SUBAPPLICATION Uebung_070 (* WBSD auf UT ausgeben *)
  (* Standard: 61499-2; Description: Copyright (c) 2023 Meisterschulen am Ostbahnhof This program and the accompanying materials are made available under the terms of the Eclipse Public License 2.0 which is available at https://www.eclipse.org/legal/epl-2.0/ SPDX-License-Identifier: EPL-2.0 *)
  (* Version 1.0, 2023-10-23, Franz Höpfinger, Meisterschulen am Ostbahnhof *)
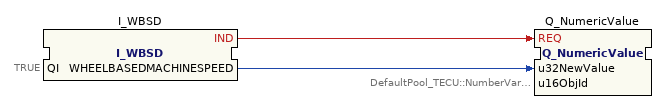
  FBS
    I_WBSD : isobus::tecu::I_WBSD(QI := TRUE);
    Q_NumericValue : isobus::ut::Q_NumericValue(u16ObjId := DefaultPool_TECU::NumberVariable_Wheel_based_machine_speed);
  END_FBS
  EVENT_CONNECTIONS
    I_WBSD.IND TO Q_NumericValue.REQ;
  END_CONNECTIONS
  DATA_CONNECTIONS
    I_WBSD.WHEELBASEDMACHINESPEED TO Q_NumericValue.u32NewValue;
  END_CONNECTIONS
END_SUBAPPLICATION
